PROGRAM TESTS
VAR
  DateTime_TEST : DateTime_TEST;
  HelperFunctions_TEST : ConvertAnyToString_TEST;
  DynamicStringBuffer_TEST : DynamicStringBuffer_TEST;
  TestWrapper : TestWrapper_NET();
END_VAR

TcUnit.RUN();

TestWrapper();

END_PROGRAM

(* stored: Version 1.1.0.1
   POU TESTS: Id {9fa91a1a-0294-47df-b5f4-55b91ebaa63a}, SpecialFunc None *)
